{attribute 'qualified_only'}
VAR_GLOBAL
END_VAR

(* stored: Version 1.1.0.1, ProductVersion 3.1.4022.7
   GVL GVL_02_Parameter_Output: Id {cf213c51-7090-4685-a7f3-e6ede36159d2} *)
